FUNCTION TryConvert_DATE_TO_UDINT : BOOL
VAR_INPUT
	in : DATE;
	out : REFERENCE TO UDINT;
END_VAR

out := DATE_TO_UDINT(in);
TryConvert_DATE_TO_UDINT := TRUE;

END_FUNCTION

(* stored: Version 1.1.0.1, ProductVersion 3.1.4024.12
   POU TryConvert_DATE_TO_UDINT: Id {e1aea9b3-02ab-4e71-8d30-dbbd4d51bb73}, SpecialFunc None *)
